Universal Robots PolyScope program: testhomeang.urp

Program testhomeang (installation=robot2 directory=/programs createdIn=5.21.3 lastSavedIn=5.21.3 robotSerialNumber=20246801938)
Calibrated DH parameters: a=[-0.000071, -0.790281, -0.600694, 0.000061, -0.000039, 0]; d=[0.236272, 604.465945, 132.116513, -736.382239, 0.159268, 0.154005]; alpha=[1.570254, -0.000567, 0.000559, 1.571709, -1.56999, 0]; deltaTheta=[0, -0.409357, 7.293326, -0.600784, -0.000001, -0.000001]
InitVariablesNode
Robot Program (runOnlyOnce=false)
  MoveL speed 250 mm/s, acceleration 1200 mm/s^2 (useActiveTCP=true optimoveEnabled=false optiMoveSpeed=0.3 optiMoveAcceleration=0.09) feature=Base
    Waypoint Waypoint_1: TCP in base x=-978.835 y=151.804 z=513.157 mm, rx=1.446 ry=-0.8 rz=-0.733 rad; joints [-48.594, -81.744, 114.027, -19.52, 7.886, -10.938] deg; TCP offset x=0.14 y=-17.51 z=284 mm, rx=0 ry=0 rz=0 rad
    Waypoint Waypoint_2: TCP in base x=-978.831 y=151.793 z=513.153 mm, rx=0.626 ry=-1.993 rz=-1.813 rad; joints [0.737, -80.947, 110.184, -18.642, 146.742, 7.644] deg
